INTERFACE ITF_GroupE_TE1_HMI EXTENDS ITF_BaseGroupElement_HMI

METHOD LinkGroupEData : BOOL
VAR_INPUT
	stData				: REFERENCE TO ST_GroupE_TE1_HMI_Link;
END_VAR
END_METHOD

END_INTERFACE

(* stored: Version 1.1.0.1, ProductVersion 3.1.4024.15
   Itf ITF_GroupE_TE1_HMI: Id {ea6c969d-098c-4608-a5ae-80f802acd029}
   Method LinkGroupEData: Id {914e8e62-c60f-492c-a283-a4d40314ad3f} *)
